FUNCTION_BLOCK FB_PrensarRodamiento_SFC
VAR_INPUT
    // SFC-Flags
    SFCPause: BOOL;
    SFCReset: BOOL;
    
    // Indicadores de sincronizacion
    Ack: BOOL := TRUE;
    Execute: BOOL;
    
    // Parametros
    RodamientoBajo: BOOL;
    TpoPrensaHidraulico: TIME := T#2S;
    TpoPrensaProtector: TIME := T#2S;
    
    // Entradas
    IntroductorDetras: BOOL := TRUE;
    IntroductorDelante: BOOL;
    ExtractorDetras: BOOL := TRUE;
    ExtractorDelante: BOOL;
    ProtectorAbajo: BOOL;
    PrensadorArriba: BOOL := TRUE;
    PrensadorAbajoAlto: BOOL;
    PrensadorAbajoBajo: BOOL;
END_VAR
VAR_OUTPUT
    // Indicadores de sincronizacion
    Done: BOOL;
    Ready: BOOL;
    
    // Salidas especificas
    IntroductorAdelante: BOOL;
    ExtractorAdelante: BOOL;
    ProtectorBaja: BOOL;
    PrensadorBaja: BOOL;
    PrensadorSube: BOOL;
    HidraulicoActiva: BOOL;
END_VAR
VAR
END_VAR

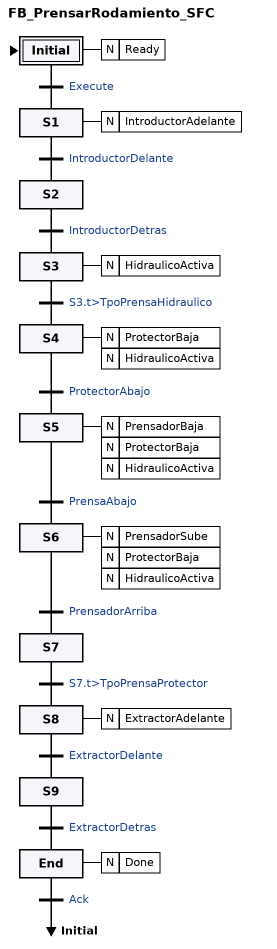
INITIAL_STEP Initial:
    Ready(N);
END_STEP
TRANSITION FROM Initial TO S1
    := Execute;
END_TRANSITION
STEP S1:
    IntroductorAdelante(N);
END_STEP
TRANSITION FROM S1 TO S2
    := IntroductorDelante;
END_TRANSITION
STEP S2:
END_STEP
TRANSITION FROM S2 TO S3
    := IntroductorDetras;
END_TRANSITION
STEP S3:
    HidraulicoActiva(N);
END_STEP
TRANSITION FROM S3 TO S4
    := S3.t>TpoPrensaHidraulico;
END_TRANSITION
STEP S4:
    ProtectorBaja(N);
    HidraulicoActiva(N);
END_STEP
TRANSITION FROM S4 TO S5
    := ProtectorAbajo;
END_TRANSITION
STEP S5:
    PrensadorBaja(N);
    ProtectorBaja(N);
    HidraulicoActiva(N);
END_STEP
TRANSITION FROM S5 TO S6
    := PrensaAbajo;
END_TRANSITION
STEP S6:
    PrensadorSube(N);
    ProtectorBaja(N);
    HidraulicoActiva(N);
END_STEP
TRANSITION FROM S6 TO S7
    := PrensadorArriba;
END_TRANSITION
STEP S7:
END_STEP
TRANSITION FROM S7 TO S8
    := S7.t>TpoPrensaProtector;
END_TRANSITION
STEP S8:
    ExtractorAdelante(N);
END_STEP
TRANSITION FROM S8 TO S9
    := ExtractorDelante;
END_TRANSITION
STEP S9:
END_STEP
TRANSITION FROM S9 TO End
    := ExtractorDetras;
END_TRANSITION
STEP End:
    Done(N);
END_STEP
TRANSITION FROM End TO Initial
    := Ack;
END_TRANSITION

TRANSITION PrensaAbajo:
// La prensa baja mas o menos dependiendo del tipo de rodamiento
(NOT RodamientoBajo AND PrensadorAbajoAlto) OR (RodamientoBajo AND PrensadorAbajoBajo)
END_TRANSITION

END_FUNCTION_BLOCK

(* stored: Version 1.1.0.1, ProductVersion 3.1.4024.12
   POU FB_PrensarRodamiento_SFC: Id {8ffd4a17-0251-484e-93ad-5050b13dbcb4}, SpecialFunc None
   Transition PrensaAbajo: Id {622623f7-fe40-46ae-a979-f74f756b34c5} *)
